TYPE DUT_VisionRegister EXTENDS DUT_StoredPosition :
STRUCT
	Scaling: REAL;
END_STRUCT
END_TYPE

(* stored: Version 1.1.0.1
   DUT DUT_VisionRegister: Id {183abbbc-75ca-4f97-a156-9832c2bf8b79} *)
